// TIA Portal V20 export
FUNCTION_BLOCK "process"   // FB1, LAD
// stored: MemoryReserve 100, Namespace ELY_1, SetENOAutomatically false
   VAR_INPUT
      Done : Bool;
   END_VAR
BEGIN
END_FUNCTION_BLOCK
